// TIA Portal V18 program export: 1 tag tables, 0 data types, 5 data blocks, 4 code blocks (in call order from the OBs), 0 instance data blocks

VAR_GLOBAL   // PLC tag table "Default tag table"
   Clock_Byte AT %MB0 : Byte;
   Clock_10Hz AT %M0.0 : Bool;
   Clock_5Hz AT %M0.1 : Bool;
   "Clock_2.5Hz" AT %M0.2 : Bool;
   Clock_2Hz AT %M0.3 : Bool;
   "Clock_1.25Hz" AT %M0.4 : Bool;
   Clock_1Hz AT %M0.5 : Bool;
   "Clock_0.625Hz" AT %M0.6 : Bool;
   "Clock_0.5Hz" AT %M0.7 : Bool;
END_VAR

DATA_BLOCK "Data_block_1"
{ S7_Optimized_Access := 'TRUE' }
VERSION : 0.1
NON_RETAIN
   VAR 
      Convalida_Lv1 : Bool;
      Convalida_Lv2 : Bool;
      Convalida_Lv3 : Bool;
      Disattiva : Bool;
      Selezione_modalita : Int;
      Password_1 : Array[0..15] of UInt;
      Password_2 : Array[0..15] of UInt;
      Password_3 : Array[0..15] of UInt;
      Lunghezza_Pw : Int;
      richiesta_lv1 : Bool;
      richiesta_lv2 : Bool;
      richiesta_lv3 : Bool;
   END_VAR


BEGIN
   Password_1[0] := 1;
   Password_1[1] := 2;
   Password_1[2] := 1;
   Password_1[3] := 1;
   Password_1[4] := 2;
   Password_1[5] := 0;
   Password_1[6] := 2;
   Password_1[7] := 3;
   Password_2[0] := 0;
   Password_2[1] := 4;
   Password_2[2] := 0;
   Password_2[3] := 9;
   Password_2[4] := 1;
   Password_2[5] := 9;
   Password_2[6] := 9;
   Password_2[7] := 7;
   Password_3[0] := 1;
   Password_3[1] := 2;
   Password_3[2] := 3;
   Password_3[3] := 4;
   Password_3[4] := 5;
   Password_3[5] := 6;
   Password_3[6] := 7;
   Password_3[7] := 8;
   Password_3[8] := 0;
   Password_3[9] := 0;
   Lunghezza_Pw := 8;

END_DATA_BLOCK

DATA_BLOCK "Logica_PW_DB"
{ S7_Optimized_Access := 'TRUE' }
VERSION : 0.1
NON_RETAIN
"Logica_PW"

BEGIN

END_DATA_BLOCK

DATA_BLOCK "Logica_TIP_DB"
{ S7_Optimized_Access := 'TRUE' }
VERSION : 0.1
NON_RETAIN
"Logica_TIP"

BEGIN

END_DATA_BLOCK

DATA_BLOCK "Variabili"
{ S7_Optimized_Access := 'TRUE' }
VERSION : 0.1
NON_RETAIN
   VAR 
      Array_Input : Array[0..3] of UInt;
      Conteggio : UInt;
      Risultato : UInt;
      Array_Memoria : Array[0..11] of Bool;
      Array_Fronti : Array[0..11] of Bool;
      Visibilità : Bool;
      Numero : UInt;
      Fronte_Richiesta_1 : Bool;
      Livello_1 : Bool;
      Richiesta_Lv1 : Bool;
      Fronte_Disabilità : Bool;
   END_VAR


BEGIN

END_DATA_BLOCK

DATA_BLOCK "IEC_Timer_0_DB_1"
{InstructionName := 'IEC_TIMER';
 LibVersion := '1.0';
 S7_Optimized_Access := 'TRUE' }
AUTHOR : Simatic
FAMILY : IEC
NAME : IEC_TMR
VERSION : 1.0
NON_RETAIN
IEC_TIMER

BEGIN

END_DATA_BLOCK

ORGANIZATION_BLOCK "Main"   // OB1, LAD, ProgramCycle
TITLE = "Main Program Sweep (Cycle)"
{ S7_Optimized_Access := 'TRUE' }
// stored: SetENOAutomatically false
   VAR_INPUT
      Initial_Call : Bool;   // Initial call of this OB
      Remanence : Bool;   // =True, if remanent data are available
   END_VAR
BEGIN

REGION Network 1
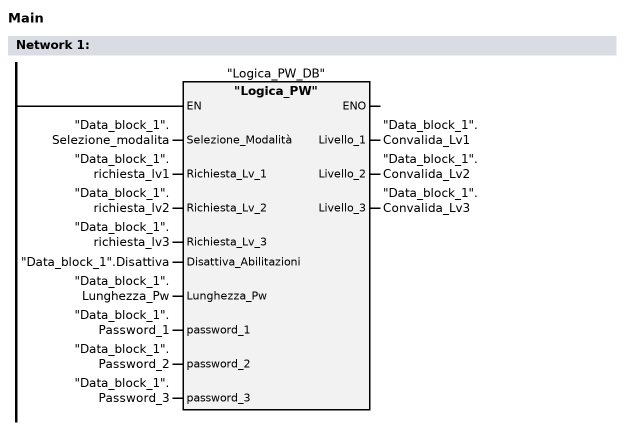
   RUNG wire#powerrail
      "Logica_PW_DB"(Selezione_Modalità := "Data_block_1".Selezione_modalita, Richiesta_Lv_1 := "Data_block_1".richiesta_lv1, Richiesta_Lv_2 := "Data_block_1".richiesta_lv2, Richiesta_Lv_3 := "Data_block_1".richiesta_lv3, Disattiva_Abilitazioni := "Data_block_1".Disattiva, Lunghezza_Pw := "Data_block_1".Lunghezza_Pw, password_1 := "Data_block_1".Password_1, password_2 := "Data_block_1".Password_2, password_3 := "Data_block_1".Password_3, Livello_1 => "Data_block_1".Convalida_Lv1, Livello_2 => "Data_block_1".Convalida_Lv2, Livello_3 => "Data_block_1".Convalida_Lv3)
   END_RUNG
   // the same network as SCL:
   "Logica_PW_DB"(Selezione_Modalità := "Data_block_1".Selezione_modalita,   // "Logica_PW"
                  Richiesta_Lv_1 := "Data_block_1".richiesta_lv1,
                  Richiesta_Lv_2 := "Data_block_1".richiesta_lv2,
                  Richiesta_Lv_3 := "Data_block_1".richiesta_lv3,
                  Disattiva_Abilitazioni := "Data_block_1".Disattiva,
                  Lunghezza_Pw := "Data_block_1".Lunghezza_Pw,
                  password_1 := "Data_block_1".Password_1,
                  password_2 := "Data_block_1".Password_2,
                  password_3 := "Data_block_1".Password_3,
                  Livello_1 => "Data_block_1".Convalida_Lv1,
                  Livello_2 => "Data_block_1".Convalida_Lv2,
                  Livello_3 => "Data_block_1".Convalida_Lv3);
END_REGION
END_ORGANIZATION_BLOCK

FUNCTION_BLOCK "Logica_PW"   // FB1, LAD
{ S7_Optimized_Access := 'TRUE' }
// stored: MemoryReserve 100, SetENOAutomatically false
   VAR_INPUT
      Selezione_Modalità { ExternalAccessible := 'False'; ExternalVisible := 'False'; ExternalWritable := 'False'} : Int;
      Richiesta_Lv_1 { ExternalAccessible := 'False'; ExternalVisible := 'False'; ExternalWritable := 'False'} : Bool;
      Richiesta_Lv_2 { ExternalAccessible := 'False'; ExternalVisible := 'False'; ExternalWritable := 'False'} : Bool;
      Richiesta_Lv_3 { ExternalAccessible := 'False'; ExternalVisible := 'False'; ExternalWritable := 'False'} : Bool;
      Disattiva_Abilitazioni { ExternalAccessible := 'False'; ExternalVisible := 'False'; ExternalWritable := 'False'} : Bool;
      Lunghezza_Pw { ExternalAccessible := 'False'; ExternalVisible := 'False'; ExternalWritable := 'False'} : Int;
   END_VAR
   VAR_OUTPUT
      Livello_1 { ExternalAccessible := 'False'; ExternalVisible := 'False'; ExternalWritable := 'False'} : Bool;
      Livello_2 { ExternalAccessible := 'False'; ExternalVisible := 'False'; ExternalWritable := 'False'} : Bool;
      Livello_3 { ExternalAccessible := 'False'; ExternalVisible := 'False'; ExternalWritable := 'False'} : Bool;
   END_VAR
   VAR_IN_OUT
      password_1 : Array[0..#N_Array] of UInt;
      password_2 : Array[0..#N_Array] of UInt;
      password_3 : Array[0..#N_Array] of UInt;
   END_VAR
   VAR
      Array_Input : Array[0..#N_Array] of UInt;
      Array_Linee : Array[0..#N_Array] of Bool;
      Conteggio : UInt;
      Risultato : UInt;
      Array_Memoria : Array[0..#N_Array] of Bool;
      Array_Fronti : Array[0..#N_Array] of Bool;
      Array_Fronti_Change : Array[0..#N_Array] of Bool;
      Visibilità : Bool;
      Numero : UInt;
      visibilità_Numeri : UInt;
      "Visibilità_Numeri_*" : UInt;
      "Visibilità_Numeri_°" : UInt;
      Fronte_Visibilità : Bool;
      Fronte_Richiesta_1 : Bool;
      Fronte_Richiesta_2 : Bool;
      Fronte_Richiesta_3 : Bool;
      Attiva_Change : Bool;
      Stato_Cambio_Pw : UInt;
      Richiesta_Lv1 : Bool;
      Richiesta_Lv2 : Bool;
      Richiesta_Lv3 : Bool;
      Fronte_Disabilità : Bool;
      Variabili_Scritte_Change : String;
      Change_Status : UInt;
      Fronte_Clock : Bool;
      "Password_Selected_ Change" : UInt;
      ET : Time;
   END_VAR
   VAR_TEMP
      n : Int;
   END_VAR
   VAR CONSTANT
      N_Array : Int := 15;
   END_VAR
   VAR_TEMP   // added for the SCL form of the ladder/FBD networks
      _w1 : Bool;
      _w2 : Bool;
      _w3 : Bool;
   END_VAR
BEGIN

REGION Network 1
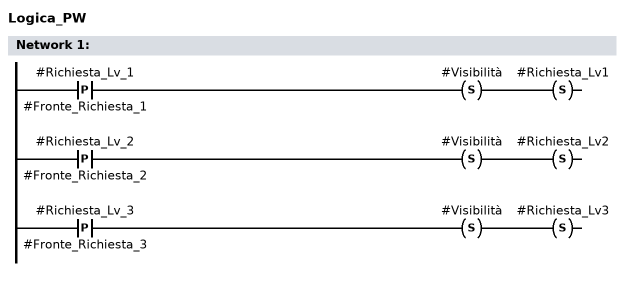
   RUNG wire#powerrail
      P_Contact(operand := #Richiesta_Lv_1, bit := #Fronte_Richiesta_1)
      S_Coil( #Visibilità )
      S_Coil( #Richiesta_Lv1 )
   END_RUNG
   RUNG wire#powerrail
      P_Contact(operand := #Richiesta_Lv_2, bit := #Fronte_Richiesta_2)
      S_Coil( #Visibilità )
      S_Coil( #Richiesta_Lv2 )
   END_RUNG
   RUNG wire#powerrail
      P_Contact(operand := #Richiesta_Lv_3, bit := #Fronte_Richiesta_3)
      S_Coil( #Visibilità )
      S_Coil( #Richiesta_Lv3 )
   END_RUNG
   // the same network as SCL:
   #_w1 := #Richiesta_Lv_1 AND NOT #Fronte_Richiesta_1;   // rising edge of #Richiesta_Lv_1
   #Fronte_Richiesta_1 := #Richiesta_Lv_1;
   IF #_w1 THEN
       #Visibilità := TRUE;
       #Richiesta_Lv1 := TRUE;
   END_IF;
   #_w2 := #Richiesta_Lv_2 AND NOT #Fronte_Richiesta_2;   // rising edge of #Richiesta_Lv_2
   #Fronte_Richiesta_2 := #Richiesta_Lv_2;
   IF #_w2 THEN
       #Visibilità := TRUE;
       #Richiesta_Lv2 := TRUE;
   END_IF;
   #_w3 := #Richiesta_Lv_3 AND NOT #Fronte_Richiesta_3;   // rising edge of #Richiesta_Lv_3
   #Fronte_Richiesta_3 := #Richiesta_Lv_3;
   IF #_w3 THEN
       #Visibilità := TRUE;
       #Richiesta_Lv3 := TRUE;
   END_IF;
END_REGION

REGION Network 2 (SCL)
   IF #Visibilità = TRUE AND #Fronte_Visibilità = false THEN
       #Variabili_Scritte_Change := 'inserisci password';
       IF #Risultato = 0 THEN  //verifico se la visibilità delle scritte è ancora a zero e nel caso la metto a 1
           #Risultato := 1;
           #visibilità_Numeri := 1;
           #Conteggio := 0;
       END_IF;
   END_IF;
   #Fronte_Visibilità := #Visibilità;
   IF #Visibilità = TRUE  THEN  //verifico se la visibilità è attiva
       REGION gestione linee e numeri/asterischi
           IF "Clock_1.25Hz" = true THEN
               #Array_Linee[#Conteggio] := true;
           ELSE
               FOR #n := 0 TO #N_Array DO
                   #Array_Linee[#n] := FALSE;
               END_FOR;
           END_IF;

           IF "Clock_10Hz" <> #Fronte_Clock THEN
               FOR #n := 0 TO #N_Array DO
                   #Array_Linee[#n] := FALSE;
               END_FOR;
           END_IF;
           #Fronte_Clock := "Clock_10Hz";


           IF #Array_Memoria[13] = true THEN
               #visibilità_Numeri := 2;
           END_IF;

           IF #Array_Memoria[13] = false & #Array_Fronti[13] = true THEN
               IF "IEC_Timer_0_DB_1".Q = true THEN
                   #visibilità_Numeri := 2;
               ELSE
                   #visibilità_Numeri := 1;
               END_IF;
           END_IF;
           #Array_Fronti[13] := #Array_Memoria[13];

           "IEC_Timer_0_DB_1".TON(IN := #Array_Memoria[13],
                                  PT := T#1s,
                                  ET => #ET);

           CASE #visibilità_Numeri OF
               1:
                   #"Visibilità_Numeri_°" := 0;
                   #"Visibilità_Numeri_*" := #Lunghezza_Pw;
               2:
                   #"Visibilità_Numeri_°" := #Lunghezza_Pw;
                   #"Visibilità_Numeri_*" := 0;
           END_CASE;
       END_REGION

       REGION rilevamento e gestione pulsanti 
           REGION rilevamento e funzionalita pulsante esc
               // pressione pulsante "ESC"
               IF (#Array_Memoria[11] = true) & (#Array_Fronti[11] = false) THEN
                   #Risultato := 1;
                   FOR #n := 0 TO #N_Array DO
                       #Array_Input[#n] := 0;
                   END_FOR;
                   FOR #n := 0 TO #N_Array DO
                       #Array_Linee[#n] := FALSE;
                   END_FOR;
                   #Conteggio := 0;
                   #Visibilità := FALSE;
                   #Richiesta_Lv1 := false;
                   #Richiesta_Lv2 := false;
                   #Richiesta_Lv3 := false;
                   #Risultato := 0;
                   #"Visibilità_Numeri_°" := 0;
                   #"Visibilità_Numeri_*" := 0;
                   #Change_Status := 0;
               END_IF;
               #Array_Fronti[11] := #Array_Memoria[11];
           END_REGION

           REGION rilevamento e funzionalità pulsante canc
               // pressione pulsante "CANC"
               IF (#Array_Memoria[12] = true) & (#Array_Fronti[12] = false) THEN
                   #Risultato := 1;
                   FOR #n := 0 TO #N_Array DO
                       #Array_Input[#n] := 0;
                   END_FOR;
                   #Conteggio := 0;
               END_IF;
               #Array_Fronti[12] := #Array_Memoria[12];
           END_REGION

           REGION rilevamento e funzionalità pulsante indietro
               // pressione pulsante indietro
               IF (#Array_Memoria[14] = true) & (#Array_Fronti[14] = false) THEN
                   IF #Conteggio > 0 THEN
                       #Conteggio := #Conteggio - 1;
                       #Array_Input[#Conteggio] := 0;
                   END_IF;
               END_IF;
               #Array_Fronti[14] := #Array_Memoria[14];
           END_REGION

           REGION rilevamento e funzionalità pulsante disattiva abilitazioni
               IF #Disattiva_Abilitazioni = true & #Fronte_Disabilità = false THEN
                   #Livello_1 := false;
                   #Livello_2 := false;
                   #Livello_3 := false;
               END_IF;
               #Fronte_Disabilità := #Disattiva_Abilitazioni;
           END_REGION
       END_REGION

       REGION rilevazione pressione pulsanti fintanto che il numero di caratteri inseriti non superi la lunghezza_pw

           IF #Conteggio < #Lunghezza_Pw THEN  //verifico se le volte in cui i numeri sono stati premuti è minore di #lunghezza_pw

               //vado a registrare gli input dei pulsanti numerici
               IF (#Array_Memoria[0] = true) & (#Array_Fronti[0] = false) THEN
                   #Array_Linee[#Numero] := FALSE;
                   #Array_Input[#Conteggio] := 0;
                   #Conteggio := #Conteggio + 1;
               END_IF;

               #Array_Fronti[0] := #Array_Memoria[0];

               IF (#Array_Memoria[1] = true) & (#Array_Fronti[1] = false) THEN
                   #Array_Linee[#Numero] := FALSE;
                   #Array_Input[#Conteggio] := 1;
                   #Conteggio := #Conteggio + 1;
               END_IF;
               #Array_Fronti[1] := #Array_Memoria[1];

               IF (#Array_Memoria[2] = true) & (#Array_Fronti[2] = false) THEN
                   #Array_Linee[#Numero] := FALSE;
                   #Array_Input[#Conteggio] := 2;
                   #Conteggio := #Conteggio + 1;
               END_IF;
               #Array_Fronti[2] := #Array_Memoria[2];

               IF (#Array_Memoria[3] = true) & (#Array_Fronti[3] = false) THEN
                   #Array_Linee[#Numero] := FALSE;
                   #Array_Input[#Conteggio] := 3;
                   #Conteggio := #Conteggio + 1;
               END_IF;
               #Array_Fronti[3] := #Array_Memoria[3];

               IF (#Array_Memoria[4] = true) & (#Array_Fronti[4] = false) THEN
                   #Array_Linee[#Numero] := FALSE;
                   #Array_Input[#Conteggio] := 4;
                   #Conteggio := #Conteggio + 1;
               END_IF;
               #Array_Fronti[4] := #Array_Memoria[4];

               IF (#Array_Memoria[5] = true) & (#Array_Fronti[5] = false) THEN
                   #Array_Linee[#Numero] := FALSE;
                   #Array_Input[#Conteggio] := 5;
                   #Conteggio := #Conteggio + 1;
               END_IF;
               #Array_Fronti[5] := #Array_Memoria[5];

               IF (#Array_Memoria[6] = true) & (#Array_Fronti[6] = false) THEN
                   #Array_Linee[#Numero] := FALSE;
                   #Array_Input[#Conteggio] := 6;
                   #Conteggio := #Conteggio + 1;
               END_IF;
               #Array_Fronti[6] := #Array_Memoria[6];

               IF (#Array_Memoria[7] = true) & (#Array_Fronti[7] = false) THEN
                   #Array_Linee[#Numero] := FALSE;
                   #Array_Input[#Conteggio] := 7;
                   #Conteggio := #Conteggio + 1;
               END_IF;
               #Array_Fronti[7] := #Array_Memoria[7];

               IF (#Array_Memoria[8] = true) & (#Array_Fronti[8] = false) THEN
                   #Array_Linee[#Numero] := FALSE;
                   #Array_Input[#Conteggio] := 8;
                   #Conteggio := #Conteggio + 1;
               END_IF;
               #Array_Fronti[8] := #Array_Memoria[8];

               IF (#Array_Memoria[9] = true) & (#Array_Fronti[9] = false) THEN
                   #Array_Linee[#Numero] := FALSE;
                   #Array_Input[#Conteggio] := 9;
                   #Conteggio := #Conteggio + 1;
               END_IF;
               #Array_Fronti[9] := #Array_Memoria[9];
           END_IF;
       END_REGION

       REGION Change_Status=0
           IF #Change_Status = 0 THEN

               REGION Restituzione risultato in base alla MODalità di funzionamento selezionata

                   IF (#Array_Memoria[10] = true) & (#Array_Fronti[10] = false) THEN
                       CASE #Selezione_Modalità OF
                           0:
                               IF #Array_Input = #password_1 THEN
                                   #Risultato := 2;
                                   #Livello_1 := true;
                                   #Livello_2 := true;
                                   #Livello_3 := true;
                                   #Variabili_Scritte_Change := 'Password corretta';
                               ELSE
                                   IF #Array_Input = #password_2 THEN
                                       #Risultato := 2;
                                       #Livello_2 := true;
                                       #Livello_3 := true;
                                       #Variabili_Scritte_Change := 'Password corretta';
                                   ELSE
                                       IF #Array_Input = #password_3 THEN
                                           #Risultato := 2;
                                           #Livello_3 := true;
                                           #Variabili_Scritte_Change := 'Password corretta';
                                       ELSE
                                           #Risultato := 3;
                                           #Variabili_Scritte_Change := 'Password sbagliata';
                                       END_IF;
                                   END_IF;
                               END_IF;
                           1:
                               IF #Richiesta_Lv1 = true THEN
                                   IF #Array_Input = #password_1 THEN
                                       #Risultato:= 2;
                                       #Livello_1 := true;
                                   ELSE
                                       #Risultato := 3;
                                   END_IF;
                               END_IF;
                               IF #Richiesta_Lv2 = true THEN
                                   IF #Array_Input = #password_2 THEN
                                       #Risultato := 2;
                                       #Livello_2 := true;
                                   ELSE
                                     #Risultato := 3;
                                   END_IF;
                               END_IF;
                               IF #Richiesta_Lv3 = true THEN
                                   IF #Array_Input = #password_3 THEN
                                       #Risultato := 2;
                                       #Livello_3 := true;
                                   ELSE
                                       #Risultato := 3;
                                   END_IF;
                               END_IF;
                           2:
                               IF #Array_Input = #password_1 THEN
                                  #Risultato := 2;
                                   #Livello_1:= true;
                                   #Livello_2:= true;
                                   #Livello_3 := true;
                               ELSE
                                   #Risultato := 3;
                               END_IF;
                       END_CASE;
                   END_IF;
                   #Array_Fronti[10] := #Array_Memoria[10];

               END_REGION

           END_IF;

       END_REGION

       REGION gestione modalità cambio password

           REGION Pressione pulsante change password ed entrata nella modalità sovrascrittura
               IF (#Array_Memoria[15] = true) & (#Array_Fronti[15] = false) THEN
                   #Variabili_Scritte_Change := 'Seleziona password da modificare';
                   FOR #n := 0 TO #N_Array DO
                       #Array_Input[#n] := 0;
                   END_FOR;
                   #Conteggio := 0;
                   #Change_Status := 1;
               END_IF;
               #Array_Fronti[15] := #Array_Memoria[15];
           END_REGION

           REGION Change_Status=1

               IF #Change_Status = 1 THEN
                   IF (#Array_Memoria[1] = true) & (#Array_Fronti_Change[1] = false) THEN
                       FOR #n := 0 TO #N_Array DO
                           #Array_Input[#n] := 0;
                       END_FOR;
                       #Conteggio := 0;
                       #Variabili_Scritte_Change := 'password precedente';
                       #Change_Status := 2;
                       #"Password_Selected_ Change" := 1;
                   END_IF;
                   #Array_Fronti_Change[1] := #Array_Memoria[1];

                   IF (#Array_Memoria[2] = true) & (#Array_Fronti_Change[2] = false) THEN
                       FOR #n := 0 TO #N_Array DO
                           #Array_Input[#n] := 0;
                       END_FOR;
                       #Conteggio := 0;
                       #Variabili_Scritte_Change :='password precedente'; // 
                       #Change_Status := 2;
                       #"Password_Selected_ Change" := 2;
                   END_IF;
                   #Array_Fronti_Change[2] := #Array_Memoria[2];


                   IF (#Array_Memoria[3] = true) & (#Array_Fronti_Change[3] = false) THEN
                       FOR #n := 0 TO #N_Array DO
                           #Array_Input[#n] := 0;
                       END_FOR;
                       #Conteggio := 0;
                       #Variabili_Scritte_Change :='password precedente';
                       #Change_Status := 2;
                       #"Password_Selected_ Change" := 3;
                   END_IF;
                   #Array_Fronti_Change[3] := #Array_Memoria[3];
               END_IF;

           END_REGION


           REGION Change_Status=2
               IF #Change_Status = 2 THEN
                   IF #Array_Memoria[10] = true & #Array_Fronti_Change[10] = FALSE THEN
                       CASE #"Password_Selected_ Change" OF
                           1:
                               IF #Array_Input = #"password_1" THEN
                                   #Change_Status := 3;
                                   FOR #n := 0 TO #N_Array DO
                                       #Array_Input[#n] := 0;
                                   END_FOR;
                                   #Conteggio := 0;
                                   #Variabili_Scritte_Change := 'Nuova password';
                               ELSE
                                   #Variabili_Scritte_Change := 'Password errata';
                               END_IF;
                           2:
                               IF #Array_Input = #password_2 THEN
                                   #Change_Status := 3;
                                   FOR #n := 0 TO #N_Array DO
                                       #Array_Input[#n] := 0;
                                   END_FOR;
                                   #Conteggio := 0;
                                   #Variabili_Scritte_Change := 'Nuova password';
                               ELSE
                                   #Variabili_Scritte_Change := 'Password errata';
                               END_IF;
                           3:
                               IF #Array_Input = #password_3 THEN
                                   #Change_Status := 3;
                                   FOR #n := 0 TO #N_Array DO
                                       #Array_Input[#n] := 0;
                                   END_FOR;
                                   #Conteggio := 0;
                                   #Variabili_Scritte_Change := 'Nuova password';
                               ELSE
                                   #Variabili_Scritte_Change := 'Password errata';
                               END_IF;
                       END_CASE;
                   END_IF;
                   #Array_Fronti_Change[10] := #Array_Memoria[10];
               END_IF;


           END_REGION


           REGION Change_Status=3
                   IF #Change_Status = 3 THEN
                       IF #Array_Memoria[10] = true & #Array_Fronti_Change[11] = FALSE THEN
                           CASE #"Password_Selected_ Change" OF
                               1:
                                   #Variabili_Scritte_Change := 'Password modificata';
                                   #"password_1" := #Array_Input;
                                   FOR #n := 0 TO #N_Array DO
                                       #Array_Input[#n] := 0;
                                   END_FOR;
                                   #Conteggio := 0;
                                   #Change_Status := 0;

                               2:
                                   #Variabili_Scritte_Change := 'Password modificata';
                                   #"password_2" := #Array_Input;
                                   FOR #n := 0 TO #N_Array DO
                                       #Array_Input[#n] := 0;
                                   END_FOR;
                                   #Conteggio := 0;
                                   #Change_Status := 0;

                               3:
                                   #Variabili_Scritte_Change := 'Password modificata';
                                   #"password_3" := #Array_Input;
                                   FOR #n := 0 TO #N_Array DO
                                       #Array_Input[#n] := 0;
                                   END_FOR;
                                   #Conteggio := 0;
                                   #Change_Status := 0;

                           END_CASE;
                       END_IF;
                       #Array_Fronti_Change[11] := #Array_Memoria[10];
                   END_IF;


               END_REGION



       END_REGION

   END_IF;
END_REGION
END_FUNCTION_BLOCK

FUNCTION "Logica" : Void   // FC1, LAD
{ S7_Optimized_Access := 'TRUE' }
// stored: AutoNumber false, SetENOAutomatically false
   VAR_INPUT
      Richiesta_Lv_1 : Bool;
      Disattiva_Abilitazioni : Bool;
      Password_1 : Array[0..3] of UInt;
   END_VAR
   VAR_OUTPUT
      Livello_1 : Bool;
   END_VAR
   VAR_TEMP   // added for the SCL form of the ladder/FBD networks
      _w1 : Bool;
   END_VAR
BEGIN

REGION Network 1
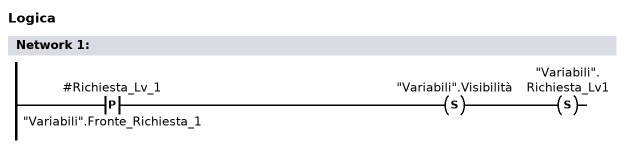
   RUNG wire#powerrail
      P_Contact(operand := #Richiesta_Lv_1, bit := "Variabili".Fronte_Richiesta_1)
      S_Coil( "Variabili".Visibilità )
      S_Coil( "Variabili".Richiesta_Lv1 )
   END_RUNG
   // the same network as SCL:
   #_w1 := #Richiesta_Lv_1 AND NOT "Variabili".Fronte_Richiesta_1;   // rising edge of #Richiesta_Lv_1
   "Variabili".Fronte_Richiesta_1 := #Richiesta_Lv_1;
   IF #_w1 THEN
       "Variabili".Visibilità := TRUE;
       "Variabili".Richiesta_Lv1 := TRUE;
   END_IF;
END_REGION

REGION Network 2 (SCL)
   IF "Variabili".Visibilità = TRUE THEN  //verifico se la visibilità è attiva
       IF "Variabili".Risultato = 0 THEN
             "Variabili".Risultato := 1;
         END_IF;

       IF "Variabili".Conteggio < 4 THEN  //verifico se le volte in cui i numeri sono stati premuti è minore di 4
           //vado a registrare gli input dei pulsanti numerici
           IF ("Variabili".Array_Memoria[0] = true) & ("Variabili".Array_Fronti[0] = false) THEN
                 "Variabili".Array_Input["Variabili".Conteggio] := 0;
                 "Variabili".Conteggio := "Variabili".Conteggio + 1;
             END_IF;

           IF ("Variabili".Array_Memoria[1] = true) & ("Variabili".Array_Fronti[1] = false) THEN
                 "Variabili".Array_Input["Variabili".Conteggio] := 1;
                 "Variabili".Conteggio := "Variabili".Conteggio + 1;
             END_IF;

           IF ("Variabili".Array_Memoria[2] = true) & ("Variabili".Array_Fronti[2] = false) THEN
                 "Variabili".Array_Input["Variabili".Conteggio] := 2;
                 "Variabili".Conteggio := "Variabili".Conteggio + 1;
             END_IF;

           IF ("Variabili".Array_Memoria[3] = true) & ("Variabili".Array_Fronti[3] = false) THEN
                 "Variabili".Array_Input["Variabili".Conteggio] := 3;
                 "Variabili".Conteggio := "Variabili".Conteggio + 1;
             END_IF;

           IF ("Variabili".Array_Memoria[4] = true) & ("Variabili".Array_Fronti[4] = false) THEN
                 "Variabili".Array_Input["Variabili".Conteggio] := 4;
                 "Variabili".Conteggio := "Variabili".Conteggio + 1;
           END_IF;

           IF ("Variabili".Array_Memoria[5] = true) & ("Variabili".Array_Fronti[5] = false) THEN
                 "Variabili".Array_Input["Variabili".Conteggio] := 5;
                 "Variabili".Conteggio := "Variabili".Conteggio + 1;
             END_IF;

           IF ("Variabili".Array_Memoria[6] = true) & ("Variabili".Array_Fronti[6] = false) THEN
                 "Variabili".Array_Input["Variabili".Conteggio] := 6;
                 "Variabili".Conteggio := "Variabili".Conteggio + 1;
             END_IF;

           IF ("Variabili".Array_Memoria[7] = true) & ("Variabili".Array_Fronti[7] = false) THEN
                 "Variabili".Array_Input["Variabili".Conteggio] := 7;
                 "Variabili".Conteggio := "Variabili".Conteggio + 1;
           END_IF;

           IF ("Variabili".Array_Memoria[8] = true) & ("Variabili".Array_Fronti[8] = false) THEN
                 "Variabili".Array_Input["Variabili".Conteggio] := 8;
                 "Variabili".Conteggio := "Variabili".Conteggio + 1;
             END_IF;

           IF ("Variabili".Array_Memoria[9] = true) & ("Variabili".Array_Fronti[9] = false) THEN
                 "Variabili".Array_Input["Variabili".Conteggio] := 9;
                 "Variabili".Conteggio := "Variabili".Conteggio + 1;
           END_IF;

       END_IF;

       IF ("Variabili".Array_Memoria[10] = true) & ("Variabili".Array_Fronti[10] = false) THEN
                   IF "Variabili".Array_Input = #Password_1 THEN
                         "Variabili".Risultato := 2;
                         "Variabili".Livello_1 := true;
                   ELSE
                         "Variabili".Risultato := 3;
                   END_IF;
       END_IF;

       // pressione pulsante "ESC"
       IF ("Variabili".Array_Memoria[11] = true) & ("Variabili".Array_Fronti[11] = false) THEN
            FOR "Variabili".Numero := 0 TO 11 DO
                  "Variabili".Array_Input["Variabili".Numero] := 0;
            END_FOR;
            "Variabili".Conteggio := 0;
            "Variabili".Risultato := 0;
            "Variabili".Visibilità := FALSE;
            "Variabili".Richiesta_Lv1 := false;
       END_IF;

   END_IF;

   IF "Variabili".Livello_1 = true THEN
       #Livello_1 := true;
   END_IF;

   IF #Disattiva_Abilitazioni = true & "Variabili".Fronte_Disabilità = false THEN
       "Variabili".Livello_1 := false;
   END_IF;


   "Variabili".Array_Fronti[0] := "Variabili".Array_Memoria[0];
   "Variabili".Array_Fronti[1] := "Variabili".Array_Memoria[1];
   "Variabili".Array_Fronti[2] := "Variabili".Array_Memoria[2];
   "Variabili".Array_Fronti[3] := "Variabili".Array_Memoria[3];
   "Variabili".Array_Fronti[4] := "Variabili".Array_Memoria[4];
   "Variabili".Array_Fronti[5] := "Variabili".Array_Memoria[5];
   "Variabili".Array_Fronti[6] := "Variabili".Array_Memoria[6];
   "Variabili".Array_Fronti[7] := "Variabili".Array_Memoria[7];
   "Variabili".Array_Fronti[8] := "Variabili".Array_Memoria[8];
   "Variabili".Array_Fronti[9] := "Variabili".Array_Memoria[9];
   "Variabili".Array_Fronti[10] := "Variabili".Array_Memoria[10];
   "Variabili".Array_Fronti[11] := "Variabili".Array_Memoria[11];
   "Variabili".Fronte_Disabilità := #Disattiva_Abilitazioni;
END_REGION
END_FUNCTION

FUNCTION_BLOCK "Logica_TIP"
{ S7_Optimized_Access := 'TRUE' }
VERSION : 0.1
   VAR_INPUT 
      Selezione_Modalità { ExternalAccessible := 'False'; ExternalVisible := 'False'; ExternalWritable := 'False'} : Int;
      Richiesta_Lv_1 { ExternalAccessible := 'False'; ExternalVisible := 'False'; ExternalWritable := 'False'} : Bool;
      Richiesta_Lv_2 { ExternalAccessible := 'False'; ExternalVisible := 'False'; ExternalWritable := 'False'} : Bool;
      Richiesta_Lv_3 { ExternalAccessible := 'False'; ExternalVisible := 'False'; ExternalWritable := 'False'} : Bool;
      Disattiva_Abilitazioni { ExternalAccessible := 'False'; ExternalVisible := 'False'; ExternalWritable := 'False'} : Bool;
   END_VAR

   VAR_OUTPUT 
      Livello_1 { ExternalAccessible := 'False'; ExternalVisible := 'False'; ExternalWritable := 'False'} : Bool;
      Livello_2 { ExternalAccessible := 'False'; ExternalVisible := 'False'; ExternalWritable := 'False'} : Bool;
      Livello_3 { ExternalAccessible := 'False'; ExternalVisible := 'False'; ExternalWritable := 'False'} : Bool;
   END_VAR

   VAR_IN_OUT 
      password_1 : Array[0..#N_Array] of UInt;
      password_2 : Array[0..#N_Array] of UInt;
      password_3 : Array[0..#N_Array] of UInt;
      Lunghezza_Pw { ExternalAccessible := 'False'; ExternalVisible := 'False'; ExternalWritable := 'False'} : Int;
   END_VAR

   VAR 
      Array_Input : Array[0..#N_Array] of UInt;
      Array_Linee : Array[0..#N_Array] of Bool;
      Conteggio : UInt;
      Array_Memoria : Array[0..#N_Array] of Bool;
      Array_Fronti : Array[0..#N_Array] of Bool;
      Array_Fronti_Change : Array[0..#N_Array] of Bool;
      Visibilità : Bool;
      Numero : UInt;
      visibilità_Numeri : UInt;
      "Visibilità_Numeri_*" : UInt;
      "Visibilità_Numeri_°" : UInt;
      Attiva_Change : Bool;
      Stato_Cambio_Pw : UInt;
      Richiesta_Lv1 : Bool;
      Richiesta_Lv2 : Bool;
      Richiesta_Lv3 : Bool;
      Fronte_Disabilità : Bool;
      Variabili_Scritte_Change : String;
      Change_Status : UInt;
      "Password_Selected_ Change" : UInt;
      ET : Time;
      ET_1 : Time;
      appoggio_fronte_10 : Bool;
      n_div : Array[0..10] of Int;
      Scritte_Errori : String;
      vis_Scritte_Errori : Bool;
      R1 {InstructionName := 'R_TRIG'; LibVersion := '1.0'} : R_TRIG;
      R2 {InstructionName := 'R_TRIG'; LibVersion := '1.0'} : R_TRIG;
      R3 {InstructionName := 'R_TRIG'; LibVersion := '1.0'} : R_TRIG;
      R4 {InstructionName := 'R_TRIG'; LibVersion := '1.0'} : R_TRIG;
      R5 {InstructionName := 'R_TRIG'; LibVersion := '1.0'} : R_TRIG;
      F_13 {InstructionName := 'F_TRIG'; LibVersion := '1.0'} : F_TRIG;
      R_11 {InstructionName := 'R_TRIG'; LibVersion := '1.0'} : R_TRIG;
      R_12 {InstructionName := 'R_TRIG'; LibVersion := '1.0'} : R_TRIG;
      R_14 {InstructionName := 'R_TRIG'; LibVersion := '1.0'} : R_TRIG;
      R_0 {InstructionName := 'R_TRIG'; LibVersion := '1.0'} : R_TRIG;
      R_1 {InstructionName := 'R_TRIG'; LibVersion := '1.0'} : R_TRIG;
      R_3 {InstructionName := 'R_TRIG'; LibVersion := '1.0'} : R_TRIG;
      R_4 {InstructionName := 'R_TRIG'; LibVersion := '1.0'} : R_TRIG;
      R_5 {InstructionName := 'R_TRIG'; LibVersion := '1.0'} : R_TRIG;
      R_6 {InstructionName := 'R_TRIG'; LibVersion := '1.0'} : R_TRIG;
      R_2 {InstructionName := 'R_TRIG'; LibVersion := '1.0'} : R_TRIG;
      R_7 {InstructionName := 'R_TRIG'; LibVersion := '1.0'} : R_TRIG;
      R_8 {InstructionName := 'R_TRIG'; LibVersion := '1.0'} : R_TRIG;
      R_9 {InstructionName := 'R_TRIG'; LibVersion := '1.0'} : R_TRIG;
   END_VAR

   VAR_TEMP 
      n : Int;
   END_VAR

   VAR CONSTANT 
      N_Array : Int := 15;
   END_VAR


BEGIN
	IF #Lunghezza_Pw > 16 THEN
	    #Lunghezza_Pw := 16;
	    #Scritte_Errori := 'Valore massimo inseribile: 16';
	    #vis_Scritte_Errori := true;
	END_IF;
	
	REGION monitoro le richieste abilitazioni e attivo i vari settaggi
	    #R1(CLK:=#Richiesta_Lv_1);
	    #R2(CLK:=#Richiesta_Lv_2);
	    #R3(CLK:=#Richiesta_Lv_3);
	    
	    IF #R1.Q THEN
	        #Visibilità := true;
	        #Richiesta_Lv1 := true;
	    END_IF;
	    
	    IF #R2.Q THEN
	        #Visibilità := true;
	        #Richiesta_Lv2 := true;
	    END_IF;
	    
	    IF #R3.Q THEN
	        #Visibilità := true;
	        #Richiesta_Lv3 := true;
	    END_IF;
	END_REGION
	
	REGION Gestione attivazione Visibilità
	    #R4(CLK := #Visibilità);
	    IF #R4.Q THEN
	        #Variabili_Scritte_Change := 'inserisci password';
	        #visibilità_Numeri := 1;
	        #Conteggio := 0;
	    END_IF;
	END_REGION;
	
	IF #Visibilità = TRUE THEN  //verifico se la visibilità è attiva
	    REGION gestione linee e numeri/asterischi
	        IF "Clock_1.25Hz" = true THEN
	            #Array_Linee[#Conteggio] := true;
	        ELSE
	            FOR #n := 0 TO #N_Array DO
	                #Array_Linee[#n] := FALSE;
	            END_FOR;
	        END_IF;
	        
	        #R5(CLK:="Clock_10Hz");
	        IF #R5.Q THEN
	            FOR #n := 0 TO #N_Array DO
	                #Array_Linee[#n] := FALSE;
	            END_FOR;
	        END_IF;
	        
	        #F_13(CLK:=#Array_Memoria[13]);
	        
	        IF #Array_Memoria[13] = true THEN
	            #visibilità_Numeri := 2;
	        END_IF;
	        
	        IF #F_13.Q THEN
	            IF "IEC_Timer_0_DB_1".Q = true THEN
	                #visibilità_Numeri := 2;
	            ELSE
	                #visibilità_Numeri := 1;
	            END_IF;
	        END_IF;
	    
	        
	        "IEC_Timer_0_DB_1".TON(IN := #Array_Memoria[13],
	                               PT := T#1s,
	                               ET => #ET);
	        
	        CASE #visibilità_Numeri OF
	            1:
	                #"Visibilità_Numeri_°" := 0;
	                #"Visibilità_Numeri_*" := #Lunghezza_Pw;
	            2:
	                #"Visibilità_Numeri_°" := #Lunghezza_Pw;
	                #"Visibilità_Numeri_*" := 0;
	          
	        END_CASE;
	    END_REGION
	    
	    REGION rilevamento e gestione pulsanti 
	        REGION rilevamento e funzionalita pulsante esc
	            // pressione pulsante "ESC"
	            #R_11(CLK:=#Array_Memoria[11]);
	            
	            IF #R_11.Q THEN
	                FOR #n := 0 TO #N_Array DO
	                    #Array_Input[#n] := 0;
	                END_FOR;
	                FOR #n := 0 TO #N_Array DO
	                    #Array_Linee[#n] := FALSE;
	                END_FOR;
	                #Conteggio := 0;
	                #Visibilità := FALSE;
	                #Richiesta_Lv1 := false;
	                #Richiesta_Lv2 := false;
	                #Richiesta_Lv3 := false;
	                #"Visibilità_Numeri_°" := 0;
	                #"Visibilità_Numeri_*" := 0;
	                #Change_Status := 0;
	            END_IF;
	        END_REGION
	        
	        REGION rilevamento e funzionalità pulsante canc
	            // pressione pulsante "CANC"
	            #R_12(CLK:=#Array_Memoria[12]);
	            IF #R_12.Q THEN
	                FOR #n := 0 TO #N_Array DO
	                    #Array_Input[#n] := 0;
	                END_FOR;
	                #Conteggio := 0;
	            END_IF;
	        END_REGION
	        
	        REGION rilevamento e funzionalità pulsante indietro
	            // pressione pulsante indietro
	            #R_14(CLK:=#Array_Memoria[14]);
	            IF #R_14.Q THEN
	                IF #Conteggio > 0 THEN
	                    #Conteggio := #Conteggio - 1;
	                    #Array_Input[#Conteggio] := 0;
	                END_IF;
	            END_IF;
	        END_REGION
	       
	    END_REGION
	    
	    REGION rilevazione pressione pulsanti fintanto che il numero di caratteri inseriti non superi la lunghezza_pw
	        
	        IF #Conteggio < #Lunghezza_Pw THEN  //verifico se le volte in cui i numeri sono stati premuti è minore di #lunghezza_pw
	            
	            //vado a registrare gli input dei pulsanti numerici
	            #R_0(CLK:= #Array_Memoria[0]);
	            #R_1(CLK:= #Array_Memoria[1]);
	            #R_2(CLK:= #Array_Memoria[2]);
	            #R_3(CLK:= #Array_Memoria[3]);
	            #R_4(CLK := #Array_Memoria[4]);
	            #R_5(CLK:= #Array_Memoria[5]);
	            #R_6(CLK:= #Array_Memoria[6]);
	            #R_7(CLK:= #Array_Memoria[7]);
	            #R_8(CLK:= #Array_Memoria[8]);
	            #R_9(CLK:= #Array_Memoria[9]);
	            
	            IF #R_0.Q THEN
	                #Array_Linee[#Numero] := FALSE;
	                #Array_Input[#Conteggio] := 0;
	                #Conteggio := #Conteggio + 1;
	            END_IF;
	            
	            IF #R_1.Q THEN
	                #Array_Linee[#Numero] := FALSE;
	                #Array_Input[#Conteggio] := 1;
	                #Conteggio := #Conteggio + 1;
	            END_IF;
	            
	            IF #R_2.Q  THEN
	                #Array_Linee[#Numero] := FALSE;
	                #Array_Input[#Conteggio] := 2;
	                #Conteggio := #Conteggio + 1;
	            END_IF;
	    
	            IF #R_3.Q THEN
	                #Array_Linee[#Numero] := FALSE;
	                #Array_Input[#Conteggio] := 3;
	                #Conteggio := #Conteggio + 1;
	            END_IF;
	            
	            IF #R_4.Q THEN
	                #Array_Linee[#Numero] := FALSE;
	                #Array_Input[#Conteggio] := 4;
	                #Conteggio := #Conteggio + 1;
	            END_IF;
	            
	            IF #R_5.Q THEN
	                #Array_Linee[#Numero] := FALSE;
	                #Array_Input[#Conteggio] := 5;
	                #Conteggio := #Conteggio + 1;
	            END_IF;
	            
	            IF #R_6.Q THEN
	                #Array_Linee[#Numero] := FALSE;
	                #Array_Input[#Conteggio] := 6;
	                #Conteggio := #Conteggio + 1;
	            END_IF;
	            
	            IF #R_7.Q THEN
	                #Array_Linee[#Numero] := FALSE;
	                #Array_Input[#Conteggio] := 7;
	                #Conteggio := #Conteggio + 1;
	            END_IF;
	            
	            IF #R_8.Q THEN
	                #Array_Linee[#Numero] := FALSE;
	                #Array_Input[#Conteggio] := 8;
	                #Conteggio := #Conteggio + 1;
	            END_IF;
	            
	            IF #R_9.Q THEN
	                #Array_Linee[#Numero] := FALSE;
	                #Array_Input[#Conteggio] := 9;
	                #Conteggio := #Conteggio + 1;
	            END_IF;
	
	        END_IF;
	    END_REGION
	    
	    REGION Change_Status=0
	        IF #Change_Status = 0 THEN
	            
	            REGION Restituzione risultato in base alla MODalità di funzionamento selezionata
	                
	                IF (#Array_Memoria[10] = true) & (#Array_Fronti[10] = false) THEN
	                    
	                    CASE #Selezione_Modalità OF
	                        0:
	                            FOR #n := 0 TO (#Lunghezza_Pw - 1) DO
	                                IF #Array_Input[#n] <> #password_1[#n] THEN
	                                    #n_div[0] := #n_div[0] + 1;
	                                END_IF;
	                            END_FOR;
	                            FOR #n := 0 TO (#Lunghezza_Pw - 1) DO
	                                IF #Array_Input[#n] <> #password_2[#n] THEN
	                                    #n_div[1] := #n_div[1] + 1;
	                                END_IF;
	                            END_FOR;
	                            FOR #n := 0 TO (#Lunghezza_Pw - 1) DO
	                                IF #Array_Input[#n] <> #password_3[#n] THEN
	                                    #n_div[2] := #n_div[2] + 1;
	                                END_IF;
	                            END_FOR;
	                            IF #n_div[0] = 0 THEN
	                                #Livello_1 := true;
	                                #Livello_2 := true;
	                                #Livello_3 := true;
	                                #Variabili_Scritte_Change := 'Password corretta';
	                            ELSE
	                                IF #n_div[1] = 0 THEN
	                                    #Livello_2 := true;
	                                    #Livello_3 := true;
	                                    #Variabili_Scritte_Change := 'Password corretta';
	                                ELSE
	                                    IF #n_div[2] = 0 THEN
	                                        #Livello_3 := true;
	                                        #Variabili_Scritte_Change := 'Password corretta';
	                                    ELSE
	                                        #Variabili_Scritte_Change := 'Password sbagliata';
	                                    END_IF;
	                                END_IF;
	                            END_IF;
	                            
	                                1:
	                                IF #Richiesta_Lv1 = true THEN
	                                    FOR #n := 0 TO (#Lunghezza_Pw - 1) DO
	                                        IF #Array_Input[#n] <> #password_1[#n] THEN
	                                            #n_div[3] := #n_div[3] + 1;
	                                        END_IF;
	                                    END_FOR;
	                                    IF #n_div[3] = 0 THEN
	                                        #Variabili_Scritte_Change := 'Password corretta';
	                                        #Livello_1 := true;
	                                    ELSE
	                                        #Variabili_Scritte_Change := 'Password sbagliata';
	                                    END_IF;
	                                END_IF;
	                                
	                                IF #Richiesta_Lv2 = true THEN
	                                    FOR #n := 0 TO (#Lunghezza_Pw - 1) DO
	                                        IF #Array_Input[#n] <> #password_2[#n] THEN
	                                            #n_div[4] := #n_div[4] + 1;
	                                        END_IF;
	                                    END_FOR;
	                                    IF #n_div[4] = 0 THEN
	                                        #Variabili_Scritte_Change := 'Password corretta';
	                                        #Livello_2 := true;
	                                    ELSE
	                                        #Variabili_Scritte_Change := 'Password sbagliata';
	                                    END_IF;
	                                END_IF;
	                                
	                                IF #Richiesta_Lv3 = true THEN
	                                    FOR #n := 0 TO (#Lunghezza_Pw - 1) DO
	                                        IF #Array_Input[#n] <> #password_3[#n] THEN
	                                            #n_div[5] := #n_div[5] + 1;
	                                        END_IF;
	                                    END_FOR;
	                                    IF #n_div[5] = 0 THEN
	                                        #Variabili_Scritte_Change := 'Password corretta';
	                                        #Livello_3 := true;
	                                    ELSE
	                                        #Variabili_Scritte_Change := 'Password sbagliata';
	                                    END_IF;
	                                END_IF;
	                                2:
	                                
	                                FOR #n := 0 TO (#Lunghezza_Pw - 1) DO
	                                    IF #Array_Input[#n] <> #password_1[#n] THEN
	                                        #n_div[6] := #n_div[6] + 1;
	                                    END_IF;
	                                END_FOR;
	                                IF #n_div[6] = 0 THEN
	                                    #Variabili_Scritte_Change := 'Password corretta';
	                                    #Livello_1 := true;
	                                    #Livello_2 := true;
	                                    #Livello_3 := true;
	                                ELSE
	                                    #Variabili_Scritte_Change := 'Password sbagliata';
	                                END_IF;
	                    END_CASE;
	                END_IF;
	                #Array_Fronti[10] := #Array_Memoria[10];
	                #Array_Memoria[10] := false;
	                FOR #n := 0 TO 6 DO
	                    #n_div[#n] := 0;
	                END_FOR;
	                
	            END_REGION
	            
	        END_IF;
	        
	    END_REGION
	    
	    REGION gestione modalità cambio password
	        
	        REGION Pressione pulsante change password ed entrata nella modalità sovrascrittura
	            IF (#Array_Memoria[15] = true) & (#Array_Fronti[15] = false) THEN
	                #Variabili_Scritte_Change := 'Seleziona password';
	                FOR #n := 0 TO #N_Array DO
	                    #Array_Input[#n] := 0;
	                END_FOR;
	                #Conteggio := 0;
	                #Change_Status := 1;
	            END_IF;
	            #Array_Fronti[15] := #Array_Memoria[15];
	        END_REGION
	        
	        REGION Change_Status=1
	            
	            IF #Change_Status = 1 THEN
	                IF (#Array_Memoria[1] = true) & (#Array_Fronti_Change[1] = false) THEN
	                    FOR #n := 0 TO #N_Array DO
	                        #Array_Input[#n] := 0;
	                    END_FOR;
	                    #Conteggio := 0;
	                    #Variabili_Scritte_Change := 'password precedente';
	                    #Change_Status := 2;
	                    #"Password_Selected_ Change" := 1;
	                END_IF;
	                #Array_Fronti_Change[1] := #Array_Memoria[1];
	                
	                IF (#Array_Memoria[2] = true) & (#Array_Fronti_Change[2] = false) THEN
	                    FOR #n := 0 TO #N_Array DO
	                        #Array_Input[#n] := 0;
	                    END_FOR;
	                    #Conteggio := 0;
	                    #Variabili_Scritte_Change := 'password precedente'; // 
	                    #Change_Status := 2;
	                    #"Password_Selected_ Change" := 2;
	                END_IF;
	                #Array_Fronti_Change[2] := #Array_Memoria[2];
	                
	                
	                IF (#Array_Memoria[3] = true) & (#Array_Fronti_Change[3] = false) THEN
	                    FOR #n := 0 TO #N_Array DO
	                        #Array_Input[#n] := 0;
	                    END_FOR;
	                    #Conteggio := 0;
	                    #Variabili_Scritte_Change := 'password precedente';
	                    #Change_Status := 2;
	                    #"Password_Selected_ Change" := 3;
	                END_IF;
	                #Array_Fronti_Change[3] := #Array_Memoria[3];
	            END_IF;
	            
	        END_REGION
	        
	        
	        REGION Change_Status=2
	            IF #Change_Status = 2 THEN
	                IF #Array_Memoria[10] = true & #Array_Fronti_Change[10] = FALSE THEN
	                    CASE #"Password_Selected_ Change" OF
	                        1:
	                            FOR #n := 0 TO (#Lunghezza_Pw - 1) DO
	                                IF #Array_Input[#n] <> #password_1[#n] THEN
	                                    #n_div[7] := #n_div[7] + 1;
	                                END_IF;
	                            END_FOR;
	                            IF #n_div[7] = 0  THEN
	                                #Change_Status := 3;
	                                FOR #n := 0 TO #N_Array DO
	                                    #Array_Input[#n] := 0;
	                                END_FOR;
	                                #Conteggio := 0;
	                                #Variabili_Scritte_Change := 'Nuova password';
	                                GOTO end;
	                            ELSE
	                                #Variabili_Scritte_Change := 'Password errata';
	                            END_IF;
	                            
	                        2:
	                            FOR #n := 0 TO (#Lunghezza_Pw - 1) DO
	                                IF #Array_Input[#n] <> #password_2[#n] THEN
	                                    #n_div[8] := #n_div[8] + 1;
	                                END_IF;
	                            END_FOR;
	                            IF #n_div[8] = 0 THEN
	                                #Change_Status := 3;
	                                FOR #n := 0 TO #N_Array DO
	                                    #Array_Input[#n] := 0;
	                                END_FOR;
	                                #Conteggio := 0;
	                                #Variabili_Scritte_Change := 'Nuova password';
	                                GOTO end;
	                            ELSE
	                                #Variabili_Scritte_Change := 'Password errata';
	                            END_IF;
	                        3:
	                            FOR #n := 0 TO (#Lunghezza_Pw - 1) DO
	                                IF #Array_Input[#n] <> #password_3[#n] THEN
	                                    #n_div[9] := #n_div[9] + 1;
	                                END_IF;
	                            END_FOR;
	                            IF #n_div[9] = 0 THEN
	                                #Change_Status := 3;
	                                FOR #n := 0 TO #N_Array DO
	                                    #Array_Input[#n] := 0;
	                                END_FOR;
	                                #Conteggio := 0;
	                                #Variabili_Scritte_Change := 'Nuova password';
	                                GOTO end;
	                            ELSE
	                                #Variabili_Scritte_Change := 'Password errata';
	                            END_IF;
	                    END_CASE;
	                END_IF;
	                #Array_Fronti_Change[10] := #Array_Memoria[10];
	            END_IF;
	            
	            
	        END_REGION
	        
	        
	        REGION Change_Status=3
	            IF #Change_Status = 3 THEN
	                IF #Array_Memoria[10] = true & #Array_Fronti_Change[11] = FALSE THEN
	                    #appoggio_fronte_10 := true;
	                    #Variabili_Scritte_Change := 'Password modificata';
	                END_IF;
	                "IEC_Timer_0_DB".TON(IN := #appoggio_fronte_10,
	                                     PT := T#1s,
	                                     ET => #ET_1);
	                IF "IEC_Timer_0_DB".Q = true THEN
	                    #appoggio_fronte_10 := false;
	                    CASE #"Password_Selected_ Change" OF
	                        1:
	                            #"password_1" := #Array_Input;
	                            GOTO esc;
	                        2:
	                            #"password_2" := #Array_Input;
	                            GOTO esc;
	                        3:
	                            #"password_3" := #Array_Input;
	                            GOTO esc;
	                    END_CASE;
	                esc:
	                    FOR #n := 0 TO #N_Array DO
	                        #Array_Input[#n] := 0;
	                    END_FOR;
	                    FOR #n := 0 TO #N_Array DO
	                        #Array_Linee[#n] := FALSE;
	                    END_FOR;
	                    #Conteggio := 0;
	                    #Visibilità := FALSE;
	                    #Richiesta_Lv1 := false;
	                    #Richiesta_Lv2 := false;
	                    #Richiesta_Lv3 := false;
	                    #"Visibilità_Numeri_°" := 0;
	                    #"Visibilità_Numeri_*" := 0;
	                    #Change_Status := 0;
	                END_IF;
	                #Array_Fronti_Change[11] := #Array_Memoria[10];
	                #Array_Memoria[10] := false;
	            END_IF;
	            
	            
	        END_REGION
	        
	    end:
	        #Array_Memoria[10] := false;
	        FOR #n := 7 TO 9 DO
	            #n_div[#n] := 0;
	        END_FOR;
	    END_REGION
	    
	   
	END_IF;
	
	REGION rilevamento e funzionalità pulsante disattiva abilitazioni
	    // va fuori dal controllo visibilità altrimenti non funziona
	    IF #Disattiva_Abilitazioni = true & #Fronte_Disabilità = false THEN
	        #Livello_1 := false;
	        #Livello_2 := false;
	        #Livello_3 := false;
	    END_IF;
	    #Fronte_Disabilità := #Disattiva_Abilitazioni;
	END_REGION
END_FUNCTION_BLOCK
